TYPE ST_ReloadRoundBelt_Status EXTENDS ST_StatusBasic :
STRUCT
END_STRUCT
END_TYPE

(* stored: Version 1.1.0.1, ProductVersion 3.1.4024.13
   DUT ST_ReloadRoundBelt_Status: Id {001a3803-1a62-4101-b3d8-0c8422ba0599} *)
